// TIA Portal V20 export
DATA_BLOCK "DB_OPC_Buttons"   // DB92
{ S7_Optimized_Access := 'TRUE' }
// stored: MemoryReserve 100
   VAR
      Door : "UDT_OPC_Button";
      Empty : "UDT_OPC_Button";
      Start : "UDT_OPC_Button";
      Stop : "UDT_OPC_Button";
      Powermeter { S7_SetPoint := 'True'} : "UDT_OPC_Button";
      GasAssist { S7_SetPoint := 'True'} : "UDT_OPC_Button";
      GripperUndrilledClamp : Struct
         Close : "UDT_OPC_Button";
         Open { S7_SetPoint := 'True'} : "UDT_OPC_Button";
         IsClosed { S7_SetPoint := 'True'} : Bool;
         IsOpened { S7_SetPoint := 'True'} : Bool;
      END_STRUCT;
      GripperDrilledClamp : Struct
         Close : "UDT_OPC_Button";
         Open { S7_SetPoint := 'True'} : "UDT_OPC_Button";
         IsClosed { S7_SetPoint := 'True'} : Bool;
         IsOpened { S7_SetPoint := 'True'} : Bool;
      END_STRUCT;
      SITestStop { S7_SetPoint := 'True'} : "UDT_OPC_Button";
      FixtureClamp { S7_SetPoint := 'True'} : "UDT_OPC_Button";
      FixtureVacuum { S7_SetPoint := 'True'} : "UDT_OPC_Button";
      Aspiration { S7_SetPoint := 'True'} : "UDT_OPC_Button";
      LoaderAuto { S7_SetPoint := 'True'} : "UDT_OPC_Button";
      LoaderSemiAuto { S7_SetPoint := 'True'} : "UDT_OPC_Button";
      Backlight { S7_SetPoint := 'True'} : "UDT_OPC_Button";
      ObservationCamera { S7_SetPoint := 'True'} : "UDT_OPC_Button";
      MainDoor { S7_SetPoint := 'True'} : "UDT_OPC_Button";
      WarmUp { S7_SetPoint := 'True'} : "UDT_OPC_Button";
      MachineLight { S7_SetPoint := 'True'} : "UDT_OPC_Button";
   END_VAR
BEGIN
END_DATA_BLOCK
